// Functions/Container Statistics/F_VN_MaxElementElementwise/F_VN_MaxElementElementwise_TcVnVector2_INT

	{attribute 'TcIecLibraryType'}
	{attribute 'external_name' := 'F_VN_MaxElementElementwise_TcVnVector2_INT_GUID_51ECF3A6_4E5F_DFF9_82EE_852C7A6E0756'}
	(* Gets the element wise maximum container element. *)
	FUNCTION F_VN_MaxElementElementwise_TcVnVector2_INT : HRESULT
	VAR_INPUT
		ipContainer	:	ITcVnContainer;	(* Source container *)
	END_VAR
	VAR_IN_OUT
		aMax	:	TcVnVector2_INT;	(* Returns the requested element *)
	END_VAR
	VAR_INPUT
		hrPrev	:	HRESULT;	(* HRESULT indicating the result of previous operations (If SUCCEEDED(hrPrev) equals false, no operation is executed.) *)
	END_VAR

END_FUNCTION

// Functions/Container Statistics/F_VN_MaxElementElementwise/F_VN_MaxElementElementwise_TcVnVector2_REAL

	{attribute 'TcIecLibraryType'}
	{attribute 'external_name' := 'F_VN_MaxElementElementwise_TcVnVector2_REAL_GUID_36FF9044_FDCF_D9B2_9EF3_5D22DF14193D'}
	(* Gets the element wise maximum container element. *)
	FUNCTION F_VN_MaxElementElementwise_TcVnVector2_REAL : HRESULT
	VAR_INPUT
		ipContainer	:	ITcVnContainer;	(* Source container *)
	END_VAR
	VAR_IN_OUT
		aMax	:	TcVnVector2_REAL;	(* Returns the requested element *)
	END_VAR
	VAR_INPUT
		hrPrev	:	HRESULT;	(* HRESULT indicating the result of previous operations (If SUCCEEDED(hrPrev) equals false, no operation is executed.) *)
	END_VAR

END_FUNCTION

// Functions/Container Statistics/F_VN_MaxElementElementwise/F_VN_MaxElementElementwise_TcVnVector2_SINT

	{attribute 'TcIecLibraryType'}
	{attribute 'external_name' := 'F_VN_MaxElementElementwise_TcVnVector2_SINT_GUID_B2222E5E_8B5F_D4D8_B8B7_613F506655FE'}
	(* Gets the element wise maximum container element. *)
	FUNCTION F_VN_MaxElementElementwise_TcVnVector2_SINT : HRESULT
	VAR_INPUT
		ipContainer	:	ITcVnContainer;	(* Source container *)
	END_VAR
	VAR_IN_OUT
		aMax	:	TcVnVector2_SINT;	(* Returns the requested element *)
	END_VAR
	VAR_INPUT
		hrPrev	:	HRESULT;	(* HRESULT indicating the result of previous operations (If SUCCEEDED(hrPrev) equals false, no operation is executed.) *)
	END_VAR

END_FUNCTION

// Functions/Container Statistics/F_VN_MaxElementElementwise/F_VN_MaxElementElementwise_TcVnVector2_UINT

	{attribute 'TcIecLibraryType'}
	{attribute 'external_name' := 'F_VN_MaxElementElementwise_TcVnVector2_UINT_GUID_20FFCD90_266D_DEF6_B943_7766169A45FA'}
	(* Gets the element wise maximum container element. *)
	FUNCTION F_VN_MaxElementElementwise_TcVnVector2_UINT : HRESULT
	VAR_INPUT
		ipContainer	:	ITcVnContainer;	(* Source container *)
	END_VAR
	VAR_IN_OUT
		aMax	:	TcVnVector2_UINT;	(* Returns the requested element *)
	END_VAR
	VAR_INPUT
		hrPrev	:	HRESULT;	(* HRESULT indicating the result of previous operations (If SUCCEEDED(hrPrev) equals false, no operation is executed.) *)
	END_VAR

END_FUNCTION

// Functions/Container Statistics/F_VN_MaxElementElementwise/F_VN_MaxElementElementwise_TcVnVector2_USINT

	{attribute 'TcIecLibraryType'}
	{attribute 'external_name' := 'F_VN_MaxElementElementwise_TcVnVector2_USINT_GUID_759705D1_AC56_D8D1_B875_EB16D1D15497'}
	(* Gets the element wise maximum container element. *)
	FUNCTION F_VN_MaxElementElementwise_TcVnVector2_USINT : HRESULT
	VAR_INPUT
		ipContainer	:	ITcVnContainer;	(* Source container *)
	END_VAR
	VAR_IN_OUT
		aMax	:	TcVnVector2_USINT;	(* Returns the requested element *)
	END_VAR
	VAR_INPUT
		hrPrev	:	HRESULT;	(* HRESULT indicating the result of previous operations (If SUCCEEDED(hrPrev) equals false, no operation is executed.) *)
	END_VAR

END_FUNCTION

// Functions/Container Statistics/F_VN_MaxElementElementwise/F_VN_MaxElementElementwise_TcVnVector3_INT

	{attribute 'TcIecLibraryType'}
	{attribute 'external_name' := 'F_VN_MaxElementElementwise_TcVnVector3_INT_GUID_8201BE4F_7FA6_D4DA_A679_F7186350AEF1'}
	(* Gets the element wise maximum container element. *)
	FUNCTION F_VN_MaxElementElementwise_TcVnVector3_INT : HRESULT
	VAR_INPUT
		ipContainer	:	ITcVnContainer;	(* Source container *)
	END_VAR
	VAR_IN_OUT
		aMax	:	TcVnVector3_INT;	(* Returns the requested element *)
	END_VAR
	VAR_INPUT
		hrPrev	:	HRESULT;	(* HRESULT indicating the result of previous operations (If SUCCEEDED(hrPrev) equals false, no operation is executed.) *)
	END_VAR

END_FUNCTION

// Functions/Container Statistics/F_VN_MaxElementElementwise/F_VN_MaxElementElementwise_TcVnVector3_REAL

	{attribute 'TcIecLibraryType'}
	{attribute 'external_name' := 'F_VN_MaxElementElementwise_TcVnVector3_REAL_GUID_01B744AE_DDF1_D8D6_AD1D_2564E4DF54AD'}
	(* Gets the element wise maximum container element. *)
	FUNCTION F_VN_MaxElementElementwise_TcVnVector3_REAL : HRESULT
	VAR_INPUT
		ipContainer	:	ITcVnContainer;	(* Source container *)
	END_VAR
	VAR_IN_OUT
		aMax	:	TcVnVector3_REAL;	(* Returns the requested element *)
	END_VAR
	VAR_INPUT
		hrPrev	:	HRESULT;	(* HRESULT indicating the result of previous operations (If SUCCEEDED(hrPrev) equals false, no operation is executed.) *)
	END_VAR

END_FUNCTION

// Functions/Container Statistics/F_VN_MaxElementElementwise/F_VN_MaxElementElementwise_TcVnVector3_SINT

	{attribute 'TcIecLibraryType'}
	{attribute 'external_name' := 'F_VN_MaxElementElementwise_TcVnVector3_SINT_GUID_62FCA671_CE0E_D9DF_B91A_305D94F8EDEB'}
	(* Gets the element wise maximum container element. *)
	FUNCTION F_VN_MaxElementElementwise_TcVnVector3_SINT : HRESULT
	VAR_INPUT
		ipContainer	:	ITcVnContainer;	(* Source container *)
	END_VAR
	VAR_IN_OUT
		aMax	:	TcVnVector3_SINT;	(* Returns the requested element *)
	END_VAR
	VAR_INPUT
		hrPrev	:	HRESULT;	(* HRESULT indicating the result of previous operations (If SUCCEEDED(hrPrev) equals false, no operation is executed.) *)
	END_VAR

END_FUNCTION

// Functions/Container Statistics/F_VN_MaxElementElementwise/F_VN_MaxElementElementwise_TcVnVector3_UINT

	{attribute 'TcIecLibraryType'}
	{attribute 'external_name' := 'F_VN_MaxElementElementwise_TcVnVector3_UINT_GUID_17CA3582_D75B_D4E5_96F3_81C1A0815197'}
	(* Gets the element wise maximum container element. *)
	FUNCTION F_VN_MaxElementElementwise_TcVnVector3_UINT : HRESULT
	VAR_INPUT
		ipContainer	:	ITcVnContainer;	(* Source container *)
	END_VAR
	VAR_IN_OUT
		aMax	:	TcVnVector3_UINT;	(* Returns the requested element *)
	END_VAR
	VAR_INPUT
		hrPrev	:	HRESULT;	(* HRESULT indicating the result of previous operations (If SUCCEEDED(hrPrev) equals false, no operation is executed.) *)
	END_VAR

END_FUNCTION

// Functions/Container Statistics/F_VN_MaxElementElementwise/F_VN_MaxElementElementwise_TcVnVector3_USINT

	{attribute 'TcIecLibraryType'}
	{attribute 'external_name' := 'F_VN_MaxElementElementwise_TcVnVector3_USINT_GUID_CA4AC978_BB4E_DA6E_A59D_D0FAA5AA5CC0'}
	(* Gets the element wise maximum container element. *)
	FUNCTION F_VN_MaxElementElementwise_TcVnVector3_USINT : HRESULT
	VAR_INPUT
		ipContainer	:	ITcVnContainer;	(* Source container *)
	END_VAR
	VAR_IN_OUT
		aMax	:	TcVnVector3_USINT;	(* Returns the requested element *)
	END_VAR
	VAR_INPUT
		hrPrev	:	HRESULT;	(* HRESULT indicating the result of previous operations (If SUCCEEDED(hrPrev) equals false, no operation is executed.) *)
	END_VAR

END_FUNCTION

// Functions/Container Statistics/F_VN_MaxElementElementwise/F_VN_MaxElementElementwise_TcVnVector4_DINT

	{attribute 'TcIecLibraryType'}
	{attribute 'external_name' := 'F_VN_MaxElementElementwise_TcVnVector4_DINT_GUID_CD328B5F_53BD_D10E_830D_85DBB5B313E2'}
	(* Gets the element wise maximum container element. *)
	FUNCTION F_VN_MaxElementElementwise_TcVnVector4_DINT : HRESULT
	VAR_INPUT
		ipContainer	:	ITcVnContainer;	(* Source container *)
	END_VAR
	VAR_IN_OUT
		aMax	:	TcVnVector4_DINT;	(* Returns the requested element *)
	END_VAR
	VAR_INPUT
		hrPrev	:	HRESULT;	(* HRESULT indicating the result of previous operations (If SUCCEEDED(hrPrev) equals false, no operation is executed.) *)
	END_VAR

END_FUNCTION

// Functions/Container Statistics/F_VN_MaxElementElementwise/F_VN_MaxElementElementwise_TcVnVector4_INT

	{attribute 'TcIecLibraryType'}
	{attribute 'external_name' := 'F_VN_MaxElementElementwise_TcVnVector4_INT_GUID_1F26472A_5D0C_D30F_BDCF_211A9E9155AD'}
	(* Gets the element wise maximum container element. *)
	FUNCTION F_VN_MaxElementElementwise_TcVnVector4_INT : HRESULT
	VAR_INPUT
		ipContainer	:	ITcVnContainer;	(* Source container *)
	END_VAR
	VAR_IN_OUT
		aMax	:	TcVnVector4_INT;	(* Returns the requested element *)
	END_VAR
	VAR_INPUT
		hrPrev	:	HRESULT;	(* HRESULT indicating the result of previous operations (If SUCCEEDED(hrPrev) equals false, no operation is executed.) *)
	END_VAR

END_FUNCTION

// Functions/Container Statistics/F_VN_MaxElementElementwise/F_VN_MaxElementElementwise_TcVnVector4_LREAL

	{attribute 'TcIecLibraryType'}
	{attribute 'external_name' := 'F_VN_MaxElementElementwise_TcVnVector4_LREAL_GUID_F7067E46_8455_DE11_B5D6_36771A946BF9'}
	(* Gets the element wise maximum container element. *)
	FUNCTION F_VN_MaxElementElementwise_TcVnVector4_LREAL : HRESULT
	VAR_INPUT
		ipContainer	:	ITcVnContainer;	(* Source container *)
	END_VAR
	VAR_IN_OUT
		aMax	:	TcVnVector4_LREAL;	(* Returns the requested element *)
	END_VAR
	VAR_INPUT
		hrPrev	:	HRESULT;	(* HRESULT indicating the result of previous operations (If SUCCEEDED(hrPrev) equals false, no operation is executed.) *)
	END_VAR

END_FUNCTION

// Functions/Container Statistics/F_VN_MaxElementElementwise/F_VN_MaxElementElementwise_TcVnVector4_REAL

	{attribute 'TcIecLibraryType'}
	{attribute 'external_name' := 'F_VN_MaxElementElementwise_TcVnVector4_REAL_GUID_A7B55928_9DF9_D291_8F16_9723E5982003'}
	(* Gets the element wise maximum container element. *)
	FUNCTION F_VN_MaxElementElementwise_TcVnVector4_REAL : HRESULT
	VAR_INPUT
		ipContainer	:	ITcVnContainer;	(* Source container *)
	END_VAR
	VAR_IN_OUT
		aMax	:	TcVnVector4_REAL;	(* Returns the requested element *)
	END_VAR
	VAR_INPUT
		hrPrev	:	HRESULT;	(* HRESULT indicating the result of previous operations (If SUCCEEDED(hrPrev) equals false, no operation is executed.) *)
	END_VAR

END_FUNCTION

// Functions/Container Statistics/F_VN_MaxElementElementwise/F_VN_MaxElementElementwise_TcVnVector4_SINT

	{attribute 'TcIecLibraryType'}
	{attribute 'external_name' := 'F_VN_MaxElementElementwise_TcVnVector4_SINT_GUID_BBB783C6_087A_D40B_A284_9C1E42E427DC'}
	(* Gets the element wise maximum container element. *)
	FUNCTION F_VN_MaxElementElementwise_TcVnVector4_SINT : HRESULT
	VAR_INPUT
		ipContainer	:	ITcVnContainer;	(* Source container *)
	END_VAR
	VAR_IN_OUT
		aMax	:	TcVnVector4_SINT;	(* Returns the requested element *)
	END_VAR
	VAR_INPUT
		hrPrev	:	HRESULT;	(* HRESULT indicating the result of previous operations (If SUCCEEDED(hrPrev) equals false, no operation is executed.) *)
	END_VAR

END_FUNCTION

// Functions/Container Statistics/F_VN_MaxElementElementwise/F_VN_MaxElementElementwise_TcVnVector4_UINT

	{attribute 'TcIecLibraryType'}
	{attribute 'external_name' := 'F_VN_MaxElementElementwise_TcVnVector4_UINT_GUID_65ED7CB6_2391_D985_BD33_521B77431117'}
	(* Gets the element wise maximum container element. *)
	FUNCTION F_VN_MaxElementElementwise_TcVnVector4_UINT : HRESULT
	VAR_INPUT
		ipContainer	:	ITcVnContainer;	(* Source container *)
	END_VAR
	VAR_IN_OUT
		aMax	:	TcVnVector4_UINT;	(* Returns the requested element *)
	END_VAR
	VAR_INPUT
		hrPrev	:	HRESULT;	(* HRESULT indicating the result of previous operations (If SUCCEEDED(hrPrev) equals false, no operation is executed.) *)
	END_VAR

END_FUNCTION

// Functions/Container Statistics/F_VN_MaxElementElementwise/F_VN_MaxElementElementwise_TcVnVector4_USINT

	{attribute 'TcIecLibraryType'}
	{attribute 'external_name' := 'F_VN_MaxElementElementwise_TcVnVector4_USINT_GUID_9C34A78C_F853_D377_9C12_528CEB462408'}
	(* Gets the element wise maximum container element. *)
	FUNCTION F_VN_MaxElementElementwise_TcVnVector4_USINT : HRESULT
	VAR_INPUT
		ipContainer	:	ITcVnContainer;	(* Source container *)
	END_VAR
	VAR_IN_OUT
		aMax	:	TcVnVector4_USINT;	(* Returns the requested element *)
	END_VAR
	VAR_INPUT
		hrPrev	:	HRESULT;	(* HRESULT indicating the result of previous operations (If SUCCEEDED(hrPrev) equals false, no operation is executed.) *)
	END_VAR

END_FUNCTION

// Functions/Container Statistics/F_VN_MaxElementElementwise/F_VN_MaxElementElementwise_UDINT

	{attribute 'TcIecLibraryType'}
	{attribute 'external_name' := 'F_VN_MaxElementElementwise_UDINT_GUID_2F4B8B8C_C3F6_DAC4_AE5F_3F8AE16BC0CF'}
	(* Gets the element wise maximum container element. *)
	FUNCTION F_VN_MaxElementElementwise_UDINT : HRESULT
	VAR_INPUT
		ipContainer	:	ITcVnContainer;	(* Source container *)
	END_VAR
	VAR_IN_OUT
		nMax	:	UDINT;	(* Returns the requested element *)
	END_VAR
	VAR_INPUT
		hrPrev	:	HRESULT;	(* HRESULT indicating the result of previous operations (If SUCCEEDED(hrPrev) equals false, no operation is executed.) *)
	END_VAR

END_FUNCTION

// Functions/Container Statistics/F_VN_MaxElementElementwise/F_VN_MaxElementElementwise_UINT

	{attribute 'TcIecLibraryType'}
	{attribute 'external_name' := 'F_VN_MaxElementElementwise_UINT_GUID_2C850313_EE79_D952_8816_C7A292497C14'}
	(* Gets the element wise maximum container element. *)
	FUNCTION F_VN_MaxElementElementwise_UINT : HRESULT
	VAR_INPUT
		ipContainer	:	ITcVnContainer;	(* Source container *)
	END_VAR
	VAR_IN_OUT
		nMax	:	UINT;	(* Returns the requested element *)
	END_VAR
	VAR_INPUT
		hrPrev	:	HRESULT;	(* HRESULT indicating the result of previous operations (If SUCCEEDED(hrPrev) equals false, no operation is executed.) *)
	END_VAR

END_FUNCTION

// Functions/Container Statistics/F_VN_MaxElementElementwise/F_VN_MaxElementElementwise_ULINT

	{attribute 'TcIecLibraryType'}
	{attribute 'external_name' := 'F_VN_MaxElementElementwise_ULINT_GUID_79575080_6C4D_DE0A_A408_669186C9D1B9'}
	(* Gets the element wise maximum container element. *)
	FUNCTION F_VN_MaxElementElementwise_ULINT : HRESULT
	VAR_INPUT
		ipContainer	:	ITcVnContainer;	(* Source container *)
	END_VAR
	VAR_IN_OUT
		nMax	:	ULINT;	(* Returns the requested element *)
	END_VAR
	VAR_INPUT
		hrPrev	:	HRESULT;	(* HRESULT indicating the result of previous operations (If SUCCEEDED(hrPrev) equals false, no operation is executed.) *)
	END_VAR

END_FUNCTION

// Functions/Container Statistics/F_VN_MaxElementElementwise/F_VN_MaxElementElementwise_USINT

	{attribute 'TcIecLibraryType'}
	{attribute 'external_name' := 'F_VN_MaxElementElementwise_USINT_GUID_65E5FDF1_4B0E_DAE8_B45E_43E6CAE87A8D'}
	(* Gets the element wise maximum container element. *)
	FUNCTION F_VN_MaxElementElementwise_USINT : HRESULT
	VAR_INPUT
		ipContainer	:	ITcVnContainer;	(* Source container *)
	END_VAR
	VAR_IN_OUT
		nMax	:	USINT;	(* Returns the requested element *)
	END_VAR
	VAR_INPUT
		hrPrev	:	HRESULT;	(* HRESULT indicating the result of previous operations (If SUCCEEDED(hrPrev) equals false, no operation is executed.) *)
	END_VAR

END_FUNCTION

// Functions/Container Statistics/F_VN_MedianElementElementwise/F_VN_MedianElementElementwise_DINT

	{attribute 'TcIecLibraryType'}
	{attribute 'external_name' := 'F_VN_MedianElementElementwise_DINT_GUID_29AA868C_E552_D86B_BF6B_18030732A5CC'}
	(* Gets the element wise median container element. *)
	FUNCTION F_VN_MedianElementElementwise_DINT : HRESULT
	VAR_INPUT
		ipContainer	:	ITcVnContainer;	(* Source container *)
	END_VAR
	VAR_IN_OUT
		nMedian	:	DINT;	(* Returns the requested element *)
	END_VAR
	VAR_INPUT
		hrPrev	:	HRESULT;	(* HRESULT indicating the result of previous operations (If SUCCEEDED(hrPrev) equals false, no operation is executed.) *)
	END_VAR

END_FUNCTION

// Functions/Container Statistics/F_VN_MedianElementElementwise/F_VN_MedianElementElementwise_INT

	{attribute 'TcIecLibraryType'}
	{attribute 'external_name' := 'F_VN_MedianElementElementwise_INT_GUID_CB0AC784_E2F3_DD60_B341_B4C0DD83E5BD'}
	(* Gets the element wise median container element. *)
	FUNCTION F_VN_MedianElementElementwise_INT : HRESULT
	VAR_INPUT
		ipContainer	:	ITcVnContainer;	(* Source container *)
	END_VAR
	VAR_IN_OUT
		nMedian	:	INT;	(* Returns the requested element *)
	END_VAR
	VAR_INPUT
		hrPrev	:	HRESULT;	(* HRESULT indicating the result of previous operations (If SUCCEEDED(hrPrev) equals false, no operation is executed.) *)
	END_VAR

END_FUNCTION

// Functions/Container Statistics/F_VN_MedianElementElementwise/F_VN_MedianElementElementwise_LREAL

	{attribute 'TcIecLibraryType'}
	{attribute 'external_name' := 'F_VN_MedianElementElementwise_LREAL_GUID_B5611EAF_9AFA_D3DE_9C03_D3DC20ACA830'}
	(* Gets the element wise median container element. *)
	FUNCTION F_VN_MedianElementElementwise_LREAL : HRESULT
	VAR_INPUT
		ipContainer	:	ITcVnContainer;	(* Source container *)
	END_VAR
	VAR_IN_OUT
		fMedian	:	LREAL;	(* Returns the requested element *)
	END_VAR
	VAR_INPUT
		hrPrev	:	HRESULT;	(* HRESULT indicating the result of previous operations (If SUCCEEDED(hrPrev) equals false, no operation is executed.) *)
	END_VAR

END_FUNCTION

// Functions/Container Statistics/F_VN_MedianElementElementwise/F_VN_MedianElementElementwise_REAL

	{attribute 'TcIecLibraryType'}
	{attribute 'external_name' := 'F_VN_MedianElementElementwise_REAL_GUID_21DEF917_9EFB_D3A8_BB2F_45041A3E4378'}
	(* Gets the element wise median container element. *)
	FUNCTION F_VN_MedianElementElementwise_REAL : HRESULT
	VAR_INPUT
		ipContainer	:	ITcVnContainer;	(* Source container *)
	END_VAR
	VAR_IN_OUT
		fMedian	:	REAL;	(* Returns the requested element *)
	END_VAR
	VAR_INPUT
		hrPrev	:	HRESULT;	(* HRESULT indicating the result of previous operations (If SUCCEEDED(hrPrev) equals false, no operation is executed.) *)
	END_VAR

END_FUNCTION

// Functions/Container Statistics/F_VN_MedianElementElementwise/F_VN_MedianElementElementwise_SINT

	{attribute 'TcIecLibraryType'}
	{attribute 'external_name' := 'F_VN_MedianElementElementwise_SINT_GUID_A76B5E76_04B8_D72A_96E3_B134E306B796'}
	(* Gets the element wise median container element. *)
	FUNCTION F_VN_MedianElementElementwise_SINT : HRESULT
	VAR_INPUT
		ipContainer	:	ITcVnContainer;	(* Source container *)
	END_VAR
	VAR_IN_OUT
		nMedian	:	SINT;	(* Returns the requested element *)
	END_VAR
	VAR_INPUT
		hrPrev	:	HRESULT;	(* HRESULT indicating the result of previous operations (If SUCCEEDED(hrPrev) equals false, no operation is executed.) *)
	END_VAR

END_FUNCTION

// Functions/Container Statistics/F_VN_MedianElementElementwise/F_VN_MedianElementElementwise_TcVnPoint2_DINT

	{attribute 'TcIecLibraryType'}
	{attribute 'external_name' := 'F_VN_MedianElementElementwise_TcVnPoint2_DINT_GUID_A3592C7D_4475_D8E1_B303_A13CD5FC38FB'}
	(* Gets the element wise median container element. *)
	FUNCTION F_VN_MedianElementElementwise_TcVnPoint2_DINT : HRESULT
	VAR_INPUT
		ipContainer	:	ITcVnContainer;	(* Source container *)
	END_VAR
	VAR_IN_OUT
		aMedian	:	TcVnPoint2_DINT;	(* Returns the requested element *)
	END_VAR
	VAR_INPUT
		hrPrev	:	HRESULT;	(* HRESULT indicating the result of previous operations (If SUCCEEDED(hrPrev) equals false, no operation is executed.) *)
	END_VAR

END_FUNCTION

// Functions/Container Statistics/F_VN_MedianElementElementwise/F_VN_MedianElementElementwise_TcVnPoint2_LREAL

	{attribute 'TcIecLibraryType'}
	{attribute 'external_name' := 'F_VN_MedianElementElementwise_TcVnPoint2_LREAL_GUID_58AAC7EB_5ADE_DF64_AAA7_24D37077B229'}
	(* Gets the element wise median container element. *)
	FUNCTION F_VN_MedianElementElementwise_TcVnPoint2_LREAL : HRESULT
	VAR_INPUT
		ipContainer	:	ITcVnContainer;	(* Source container *)
	END_VAR
	VAR_IN_OUT
		aMedian	:	TcVnPoint2_LREAL;	(* Returns the requested element *)
	END_VAR
	VAR_INPUT
		hrPrev	:	HRESULT;	(* HRESULT indicating the result of previous operations (If SUCCEEDED(hrPrev) equals false, no operation is executed.) *)
	END_VAR

END_FUNCTION

// Functions/Container Statistics/F_VN_MedianElementElementwise/F_VN_MedianElementElementwise_TcVnPoint2_REAL

	{attribute 'TcIecLibraryType'}
	{attribute 'external_name' := 'F_VN_MedianElementElementwise_TcVnPoint2_REAL_GUID_F85373B6_2943_D6B1_9993_6D4DB4D57329'}
	(* Gets the element wise median container element. *)
	FUNCTION F_VN_MedianElementElementwise_TcVnPoint2_REAL : HRESULT
	VAR_INPUT
		ipContainer	:	ITcVnContainer;	(* Source container *)
	END_VAR
	VAR_IN_OUT
		aMedian	:	TcVnPoint2_REAL;	(* Returns the requested element *)
	END_VAR
	VAR_INPUT
		hrPrev	:	HRESULT;	(* HRESULT indicating the result of previous operations (If SUCCEEDED(hrPrev) equals false, no operation is executed.) *)
	END_VAR

END_FUNCTION

// Functions/Container Statistics/F_VN_MedianElementElementwise/F_VN_MedianElementElementwise_TcVnPoint3_LREAL

	{attribute 'TcIecLibraryType'}
	{attribute 'external_name' := 'F_VN_MedianElementElementwise_TcVnPoint3_LREAL_GUID_F14A33BF_2275_D80A_AC45_515904B471A2'}
	(* Gets the element wise median container element. *)
	FUNCTION F_VN_MedianElementElementwise_TcVnPoint3_LREAL : HRESULT
	VAR_INPUT
		ipContainer	:	ITcVnContainer;	(* Source container *)
	END_VAR
	VAR_IN_OUT
		aMedian	:	TcVnPoint3_LREAL;	(* Returns the requested element *)
	END_VAR
	VAR_INPUT
		hrPrev	:	HRESULT;	(* HRESULT indicating the result of previous operations (If SUCCEEDED(hrPrev) equals false, no operation is executed.) *)
	END_VAR

END_FUNCTION

// Functions/Container Statistics/F_VN_MedianElementElementwise/F_VN_MedianElementElementwise_TcVnPoint3_REAL

	{attribute 'TcIecLibraryType'}
	{attribute 'external_name' := 'F_VN_MedianElementElementwise_TcVnPoint3_REAL_GUID_756F28F9_77FF_DB99_A3DB_C5C4C4331351'}
	(* Gets the element wise median container element. *)
	FUNCTION F_VN_MedianElementElementwise_TcVnPoint3_REAL : HRESULT
	VAR_INPUT
		ipContainer	:	ITcVnContainer;	(* Source container *)
	END_VAR
	VAR_IN_OUT
		aMedian	:	TcVnPoint3_REAL;	(* Returns the requested element *)
	END_VAR
	VAR_INPUT
		hrPrev	:	HRESULT;	(* HRESULT indicating the result of previous operations (If SUCCEEDED(hrPrev) equals false, no operation is executed.) *)
	END_VAR

END_FUNCTION

// Functions/Container Statistics/F_VN_MedianElementElementwise/F_VN_MedianElementElementwise_TcVnVector2_DINT

	{attribute 'TcIecLibraryType'}
	{attribute 'external_name' := 'F_VN_MedianElementElementwise_TcVnVector2_DINT_GUID_8E473526_A7CC_DFC3_9E5F_288766125041'}
	(* Gets the element wise median container element. *)
	FUNCTION F_VN_MedianElementElementwise_TcVnVector2_DINT : HRESULT
	VAR_INPUT
		ipContainer	:	ITcVnContainer;	(* Source container *)
	END_VAR
	VAR_IN_OUT
		aMedian	:	TcVnVector2_DINT;	(* Returns the requested element *)
	END_VAR
	VAR_INPUT
		hrPrev	:	HRESULT;	(* HRESULT indicating the result of previous operations (If SUCCEEDED(hrPrev) equals false, no operation is executed.) *)
	END_VAR

END_FUNCTION

// Functions/Container Statistics/F_VN_MedianElementElementwise/F_VN_MedianElementElementwise_TcVnVector2_INT

	{attribute 'TcIecLibraryType'}
	{attribute 'external_name' := 'F_VN_MedianElementElementwise_TcVnVector2_INT_GUID_5BDD346F_B29E_DEEB_A174_03D5BCDD966C'}
	(* Gets the element wise median container element. *)
	FUNCTION F_VN_MedianElementElementwise_TcVnVector2_INT : HRESULT
	VAR_INPUT
		ipContainer	:	ITcVnContainer;	(* Source container *)
	END_VAR
	VAR_IN_OUT
		aMedian	:	TcVnVector2_INT;	(* Returns the requested element *)
	END_VAR
	VAR_INPUT
		hrPrev	:	HRESULT;	(* HRESULT indicating the result of previous operations (If SUCCEEDED(hrPrev) equals false, no operation is executed.) *)
	END_VAR

END_FUNCTION

// Functions/Container Statistics/F_VN_MedianElementElementwise/F_VN_MedianElementElementwise_TcVnVector2_REAL

	{attribute 'TcIecLibraryType'}
	{attribute 'external_name' := 'F_VN_MedianElementElementwise_TcVnVector2_REAL_GUID_86E9BF9E_E3F9_D74F_9617_EB2C03F6B6E3'}
	(* Gets the element wise median container element. *)
	FUNCTION F_VN_MedianElementElementwise_TcVnVector2_REAL : HRESULT
	VAR_INPUT
		ipContainer	:	ITcVnContainer;	(* Source container *)
	END_VAR
	VAR_IN_OUT
		aMedian	:	TcVnVector2_REAL;	(* Returns the requested element *)
	END_VAR
	VAR_INPUT
		hrPrev	:	HRESULT;	(* HRESULT indicating the result of previous operations (If SUCCEEDED(hrPrev) equals false, no operation is executed.) *)
	END_VAR

END_FUNCTION

// Functions/Container Statistics/F_VN_MedianElementElementwise/F_VN_MedianElementElementwise_TcVnVector2_SINT

	{attribute 'TcIecLibraryType'}
	{attribute 'external_name' := 'F_VN_MedianElementElementwise_TcVnVector2_SINT_GUID_FF27191B_A2BB_DF95_854B_1FD1821A0F7E'}
	(* Gets the element wise median container element. *)
	FUNCTION F_VN_MedianElementElementwise_TcVnVector2_SINT : HRESULT
	VAR_INPUT
		ipContainer	:	ITcVnContainer;	(* Source container *)
	END_VAR
	VAR_IN_OUT
		aMedian	:	TcVnVector2_SINT;	(* Returns the requested element *)
	END_VAR
	VAR_INPUT
		hrPrev	:	HRESULT;	(* HRESULT indicating the result of previous operations (If SUCCEEDED(hrPrev) equals false, no operation is executed.) *)
	END_VAR

END_FUNCTION

// Functions/Container Statistics/F_VN_MedianElementElementwise/F_VN_MedianElementElementwise_TcVnVector2_UINT

	{attribute 'TcIecLibraryType'}
	{attribute 'external_name' := 'F_VN_MedianElementElementwise_TcVnVector2_UINT_GUID_705877EF_7F8F_DC5B_A99E_E66FED4F7A28'}
	(* Gets the element wise median container element. *)
	FUNCTION F_VN_MedianElementElementwise_TcVnVector2_UINT : HRESULT
	VAR_INPUT
		ipContainer	:	ITcVnContainer;	(* Source container *)
	END_VAR
	VAR_IN_OUT
		aMedian	:	TcVnVector2_UINT;	(* Returns the requested element *)
	END_VAR
	VAR_INPUT
		hrPrev	:	HRESULT;	(* HRESULT indicating the result of previous operations (If SUCCEEDED(hrPrev) equals false, no operation is executed.) *)
	END_VAR

END_FUNCTION

// Functions/Container Statistics/F_VN_MedianElementElementwise/F_VN_MedianElementElementwise_TcVnVector2_USINT

	{attribute 'TcIecLibraryType'}
	{attribute 'external_name' := 'F_VN_MedianElementElementwise_TcVnVector2_USINT_GUID_25701AD9_252E_DC2D_9926_E17D1B44381C'}
	(* Gets the element wise median container element. *)
	FUNCTION F_VN_MedianElementElementwise_TcVnVector2_USINT : HRESULT
	VAR_INPUT
		ipContainer	:	ITcVnContainer;	(* Source container *)
	END_VAR
	VAR_IN_OUT
		aMedian	:	TcVnVector2_USINT;	(* Returns the requested element *)
	END_VAR
	VAR_INPUT
		hrPrev	:	HRESULT;	(* HRESULT indicating the result of previous operations (If SUCCEEDED(hrPrev) equals false, no operation is executed.) *)
	END_VAR

END_FUNCTION

// Functions/Container Statistics/F_VN_MedianElementElementwise/F_VN_MedianElementElementwise_TcVnVector3_INT

	{attribute 'TcIecLibraryType'}
	{attribute 'external_name' := 'F_VN_MedianElementElementwise_TcVnVector3_INT_GUID_4CD6D63F_F997_D2F3_AB3B_4A33E5647F84'}
	(* Gets the element wise median container element. *)
	FUNCTION F_VN_MedianElementElementwise_TcVnVector3_INT : HRESULT
	VAR_INPUT
		ipContainer	:	ITcVnContainer;	(* Source container *)
	END_VAR
	VAR_IN_OUT
		aMedian	:	TcVnVector3_INT;	(* Returns the requested element *)
	END_VAR
	VAR_INPUT
		hrPrev	:	HRESULT;	(* HRESULT indicating the result of previous operations (If SUCCEEDED(hrPrev) equals false, no operation is executed.) *)
	END_VAR

END_FUNCTION

// Functions/Container Statistics/F_VN_MedianElementElementwise/F_VN_MedianElementElementwise_TcVnVector3_REAL

	{attribute 'TcIecLibraryType'}
	{attribute 'external_name' := 'F_VN_MedianElementElementwise_TcVnVector3_REAL_GUID_4E994DD7_D9B7_DE3E_932B_AC8B406F870C'}
	(* Gets the element wise median container element. *)
	FUNCTION F_VN_MedianElementElementwise_TcVnVector3_REAL : HRESULT
	VAR_INPUT
		ipContainer	:	ITcVnContainer;	(* Source container *)
	END_VAR
	VAR_IN_OUT
		aMedian	:	TcVnVector3_REAL;	(* Returns the requested element *)
	END_VAR
	VAR_INPUT
		hrPrev	:	HRESULT;	(* HRESULT indicating the result of previous operations (If SUCCEEDED(hrPrev) equals false, no operation is executed.) *)
	END_VAR

END_FUNCTION

// Functions/Container Statistics/F_VN_MedianElementElementwise/F_VN_MedianElementElementwise_TcVnVector3_SINT

	{attribute 'TcIecLibraryType'}
	{attribute 'external_name' := 'F_VN_MedianElementElementwise_TcVnVector3_SINT_GUID_9137D501_0F28_D22B_853D_E2549CAB39F0'}
	(* Gets the element wise median container element. *)
	FUNCTION F_VN_MedianElementElementwise_TcVnVector3_SINT : HRESULT
	VAR_INPUT
		ipContainer	:	ITcVnContainer;	(* Source container *)
	END_VAR
	VAR_IN_OUT
		aMedian	:	TcVnVector3_SINT;	(* Returns the requested element *)
	END_VAR
	VAR_INPUT
		hrPrev	:	HRESULT;	(* HRESULT indicating the result of previous operations (If SUCCEEDED(hrPrev) equals false, no operation is executed.) *)
	END_VAR

END_FUNCTION

// Functions/Container Statistics/F_VN_MedianElementElementwise/F_VN_MedianElementElementwise_TcVnVector3_UINT

	{attribute 'TcIecLibraryType'}
	{attribute 'external_name' := 'F_VN_MedianElementElementwise_TcVnVector3_UINT_GUID_A8DF8F4C_462A_D898_950A_55B3BB3E2024'}
	(* Gets the element wise median container element. *)
	FUNCTION F_VN_MedianElementElementwise_TcVnVector3_UINT : HRESULT
	VAR_INPUT
		ipContainer	:	ITcVnContainer;	(* Source container *)
	END_VAR
	VAR_IN_OUT
		aMedian	:	TcVnVector3_UINT;	(* Returns the requested element *)
	END_VAR
	VAR_INPUT
		hrPrev	:	HRESULT;	(* HRESULT indicating the result of previous operations (If SUCCEEDED(hrPrev) equals false, no operation is executed.) *)
	END_VAR

END_FUNCTION

// Functions/Container Statistics/F_VN_MedianElementElementwise/F_VN_MedianElementElementwise_TcVnVector3_USINT

	{attribute 'TcIecLibraryType'}
	{attribute 'external_name' := 'F_VN_MedianElementElementwise_TcVnVector3_USINT_GUID_0C8F98E8_0B46_D076_9A4C_AEBC34133C5E'}
	(* Gets the element wise median container element. *)
	FUNCTION F_VN_MedianElementElementwise_TcVnVector3_USINT : HRESULT
	VAR_INPUT
		ipContainer	:	ITcVnContainer;	(* Source container *)
	END_VAR
	VAR_IN_OUT
		aMedian	:	TcVnVector3_USINT;	(* Returns the requested element *)
	END_VAR
	VAR_INPUT
		hrPrev	:	HRESULT;	(* HRESULT indicating the result of previous operations (If SUCCEEDED(hrPrev) equals false, no operation is executed.) *)
	END_VAR

END_FUNCTION

// Functions/Container Statistics/F_VN_MedianElementElementwise/F_VN_MedianElementElementwise_TcVnVector4_DINT

	{attribute 'TcIecLibraryType'}
	{attribute 'external_name' := 'F_VN_MedianElementElementwise_TcVnVector4_DINT_GUID_6FADAB1A_0169_D530_9009_CC67F58ABF30'}
	(* Gets the element wise median container element. *)
	FUNCTION F_VN_MedianElementElementwise_TcVnVector4_DINT : HRESULT
	VAR_INPUT
		ipContainer	:	ITcVnContainer;	(* Source container *)
	END_VAR
	VAR_IN_OUT
		aMedian	:	TcVnVector4_DINT;	(* Returns the requested element *)
	END_VAR
	VAR_INPUT
		hrPrev	:	HRESULT;	(* HRESULT indicating the result of previous operations (If SUCCEEDED(hrPrev) equals false, no operation is executed.) *)
	END_VAR

END_FUNCTION

// Functions/Container Statistics/F_VN_MedianElementElementwise/F_VN_MedianElementElementwise_TcVnVector4_INT

	{attribute 'TcIecLibraryType'}
	{attribute 'external_name' := 'F_VN_MedianElementElementwise_TcVnVector4_INT_GUID_547BAD9B_6F7A_DD0B_8790_02EDB713B258'}
	(* Gets the element wise median container element. *)
	FUNCTION F_VN_MedianElementElementwise_TcVnVector4_INT : HRESULT
	VAR_INPUT
		ipContainer	:	ITcVnContainer;	(* Source container *)
	END_VAR
	VAR_IN_OUT
		aMedian	:	TcVnVector4_INT;	(* Returns the requested element *)
	END_VAR
	VAR_INPUT
		hrPrev	:	HRESULT;	(* HRESULT indicating the result of previous operations (If SUCCEEDED(hrPrev) equals false, no operation is executed.) *)
	END_VAR

END_FUNCTION

// Functions/Container Statistics/F_VN_MedianElementElementwise/F_VN_MedianElementElementwise_TcVnVector4_LREAL

	{attribute 'TcIecLibraryType'}
	{attribute 'external_name' := 'F_VN_MedianElementElementwise_TcVnVector4_LREAL_GUID_626602F4_5A0A_DEBF_AF13_43F5508850CD'}
	(* Gets the element wise median container element. *)
	FUNCTION F_VN_MedianElementElementwise_TcVnVector4_LREAL : HRESULT
	VAR_INPUT
		ipContainer	:	ITcVnContainer;	(* Source container *)
	END_VAR
	VAR_IN_OUT
		aMedian	:	TcVnVector4_LREAL;	(* Returns the requested element *)
	END_VAR
	VAR_INPUT
		hrPrev	:	HRESULT;	(* HRESULT indicating the result of previous operations (If SUCCEEDED(hrPrev) equals false, no operation is executed.) *)
	END_VAR

END_FUNCTION

// Functions/Container Statistics/F_VN_MedianElementElementwise/F_VN_MedianElementElementwise_TcVnVector4_REAL

	{attribute 'TcIecLibraryType'}
	{attribute 'external_name' := 'F_VN_MedianElementElementwise_TcVnVector4_REAL_GUID_49F75D51_3181_DA08_9B3B_68B99A9DF7AE'}
	(* Gets the element wise median container element. *)
	FUNCTION F_VN_MedianElementElementwise_TcVnVector4_REAL : HRESULT
	VAR_INPUT
		ipContainer	:	ITcVnContainer;	(* Source container *)
	END_VAR
	VAR_IN_OUT
		aMedian	:	TcVnVector4_REAL;	(* Returns the requested element *)
	END_VAR
	VAR_INPUT
		hrPrev	:	HRESULT;	(* HRESULT indicating the result of previous operations (If SUCCEEDED(hrPrev) equals false, no operation is executed.) *)
	END_VAR

END_FUNCTION

// Functions/Container Statistics/F_VN_MedianElementElementwise/F_VN_MedianElementElementwise_TcVnVector4_SINT

	{attribute 'TcIecLibraryType'}
	{attribute 'external_name' := 'F_VN_MedianElementElementwise_TcVnVector4_SINT_GUID_61695308_1194_D30C_87B3_CD47BB5B616F'}
	(* Gets the element wise median container element. *)
	FUNCTION F_VN_MedianElementElementwise_TcVnVector4_SINT : HRESULT
	VAR_INPUT
		ipContainer	:	ITcVnContainer;	(* Source container *)
	END_VAR
	VAR_IN_OUT
		aMedian	:	TcVnVector4_SINT;	(* Returns the requested element *)
	END_VAR
	VAR_INPUT
		hrPrev	:	HRESULT;	(* HRESULT indicating the result of previous operations (If SUCCEEDED(hrPrev) equals false, no operation is executed.) *)
	END_VAR

END_FUNCTION

// Functions/Container Statistics/F_VN_MedianElementElementwise/F_VN_MedianElementElementwise_TcVnVector4_UINT

	{attribute 'TcIecLibraryType'}
	{attribute 'external_name' := 'F_VN_MedianElementElementwise_TcVnVector4_UINT_GUID_04BDB311_7306_D375_920D_775A084C28E2'}
	(* Gets the element wise median container element. *)
	FUNCTION F_VN_MedianElementElementwise_TcVnVector4_UINT : HRESULT
	VAR_INPUT
		ipContainer	:	ITcVnContainer;	(* Source container *)
	END_VAR
	VAR_IN_OUT
		aMedian	:	TcVnVector4_UINT;	(* Returns the requested element *)
	END_VAR
	VAR_INPUT
		hrPrev	:	HRESULT;	(* HRESULT indicating the result of previous operations (If SUCCEEDED(hrPrev) equals false, no operation is executed.) *)
	END_VAR

END_FUNCTION

// Functions/Container Statistics/F_VN_MedianElementElementwise/F_VN_MedianElementElementwise_TcVnVector4_USINT

	{attribute 'TcIecLibraryType'}
	{attribute 'external_name' := 'F_VN_MedianElementElementwise_TcVnVector4_USINT_GUID_C6120573_4FCC_DD80_AD43_4ABD35A8D98B'}
	(* Gets the element wise median container element. *)
	FUNCTION F_VN_MedianElementElementwise_TcVnVector4_USINT : HRESULT
	VAR_INPUT
		ipContainer	:	ITcVnContainer;	(* Source container *)
	END_VAR
	VAR_IN_OUT
		aMedian	:	TcVnVector4_USINT;	(* Returns the requested element *)
	END_VAR
	VAR_INPUT
		hrPrev	:	HRESULT;	(* HRESULT indicating the result of previous operations (If SUCCEEDED(hrPrev) equals false, no operation is executed.) *)
	END_VAR

END_FUNCTION

// Functions/Container Statistics/F_VN_MedianElementElementwise/F_VN_MedianElementElementwise_UDINT

	{attribute 'TcIecLibraryType'}
	{attribute 'external_name' := 'F_VN_MedianElementElementwise_UDINT_GUID_9BC7BF91_3125_D729_9768_84FE886C888D'}
	(* Gets the element wise median container element. *)
	FUNCTION F_VN_MedianElementElementwise_UDINT : HRESULT
	VAR_INPUT
		ipContainer	:	ITcVnContainer;	(* Source container *)
	END_VAR
	VAR_IN_OUT
		nMedian	:	UDINT;	(* Returns the requested element *)
	END_VAR
	VAR_INPUT
		hrPrev	:	HRESULT;	(* HRESULT indicating the result of previous operations (If SUCCEEDED(hrPrev) equals false, no operation is executed.) *)
	END_VAR

END_FUNCTION

// Functions/Container Statistics/F_VN_MedianElementElementwise/F_VN_MedianElementElementwise_UINT

	{attribute 'TcIecLibraryType'}
	{attribute 'external_name' := 'F_VN_MedianElementElementwise_UINT_GUID_AA7E04F5_27DD_D1E9_89BB_71FE2A03EF73'}
	(* Gets the element wise median container element. *)
	FUNCTION F_VN_MedianElementElementwise_UINT : HRESULT
	VAR_INPUT
		ipContainer	:	ITcVnContainer;	(* Source container *)
	END_VAR
	VAR_IN_OUT
		nMedian	:	UINT;	(* Returns the requested element *)
	END_VAR
	VAR_INPUT
		hrPrev	:	HRESULT;	(* HRESULT indicating the result of previous operations (If SUCCEEDED(hrPrev) equals false, no operation is executed.) *)
	END_VAR

END_FUNCTION

// Functions/Container Statistics/F_VN_MedianElementElementwise/F_VN_MedianElementElementwise_ULINT

	{attribute 'TcIecLibraryType'}
	{attribute 'external_name' := 'F_VN_MedianElementElementwise_ULINT_GUID_8ECFBFA6_0E43_DAD1_AF9F_464DAE11C1ED'}
	(* Gets the element wise median container element. *)
	FUNCTION F_VN_MedianElementElementwise_ULINT : HRESULT
	VAR_INPUT
		ipContainer	:	ITcVnContainer;	(* Source container *)
	END_VAR
	VAR_IN_OUT
		nMedian	:	ULINT;	(* Returns the requested element *)
	END_VAR
	VAR_INPUT
		hrPrev	:	HRESULT;	(* HRESULT indicating the result of previous operations (If SUCCEEDED(hrPrev) equals false, no operation is executed.) *)
	END_VAR

END_FUNCTION

// Functions/Container Statistics/F_VN_MedianElementElementwise/F_VN_MedianElementElementwise_USINT

	{attribute 'TcIecLibraryType'}
	{attribute 'external_name' := 'F_VN_MedianElementElementwise_USINT_GUID_2994888C_8833_D8FA_BA03_E55B76F2506A'}
	(* Gets the element wise median container element. *)
	FUNCTION F_VN_MedianElementElementwise_USINT : HRESULT
	VAR_INPUT
		ipContainer	:	ITcVnContainer;	(* Source container *)
	END_VAR
	VAR_IN_OUT
		nMedian	:	USINT;	(* Returns the requested element *)
	END_VAR
	VAR_INPUT
		hrPrev	:	HRESULT;	(* HRESULT indicating the result of previous operations (If SUCCEEDED(hrPrev) equals false, no operation is executed.) *)
	END_VAR

END_FUNCTION

// Functions/Container Statistics/F_VN_MinElementElementwise/F_VN_MinElementElementwise_DINT

	{attribute 'TcIecLibraryType'}
	{attribute 'external_name' := 'F_VN_MinElementElementwise_DINT_GUID_7E567114_9BD1_D305_87D1_88AF602BEA2D'}
	(* Gets the element wise minimum container element. *)
	FUNCTION F_VN_MinElementElementwise_DINT : HRESULT
	VAR_INPUT
		ipContainer	:	ITcVnContainer;	(* Source container *)
	END_VAR
	VAR_IN_OUT
		nMin	:	DINT;	(* Returns the requested element *)
	END_VAR
	VAR_INPUT
		hrPrev	:	HRESULT;	(* HRESULT indicating the result of previous operations (If SUCCEEDED(hrPrev) equals false, no operation is executed.) *)
	END_VAR

END_FUNCTION

// Functions/Container Statistics/F_VN_MinElementElementwise/F_VN_MinElementElementwise_INT

	{attribute 'TcIecLibraryType'}
	{attribute 'external_name' := 'F_VN_MinElementElementwise_INT_GUID_0BB9518D_66CC_D115_B745_E5695DFD31B0'}
	(* Gets the element wise minimum container element. *)
	FUNCTION F_VN_MinElementElementwise_INT : HRESULT
	VAR_INPUT
		ipContainer	:	ITcVnContainer;	(* Source container *)
	END_VAR
	VAR_IN_OUT
		nMin	:	INT;	(* Returns the requested element *)
	END_VAR
	VAR_INPUT
		hrPrev	:	HRESULT;	(* HRESULT indicating the result of previous operations (If SUCCEEDED(hrPrev) equals false, no operation is executed.) *)
	END_VAR

END_FUNCTION

// Functions/Container Statistics/F_VN_MinElementElementwise/F_VN_MinElementElementwise_LREAL

	{attribute 'TcIecLibraryType'}
	{attribute 'external_name' := 'F_VN_MinElementElementwise_LREAL_GUID_C1D5880C_C085_D406_8F8C_640347E2EC83'}
	(* Gets the element wise minimum container element. *)
	FUNCTION F_VN_MinElementElementwise_LREAL : HRESULT
	VAR_INPUT
		ipContainer	:	ITcVnContainer;	(* Source container *)
	END_VAR
	VAR_IN_OUT
		fMin	:	LREAL;	(* Returns the requested element *)
	END_VAR
	VAR_INPUT
		hrPrev	:	HRESULT;	(* HRESULT indicating the result of previous operations (If SUCCEEDED(hrPrev) equals false, no operation is executed.) *)
	END_VAR

END_FUNCTION

// Functions/Container Statistics/F_VN_MinElementElementwise/F_VN_MinElementElementwise_REAL

	{attribute 'TcIecLibraryType'}
	{attribute 'external_name' := 'F_VN_MinElementElementwise_REAL_GUID_450605AD_BDF8_DB97_BA29_50E9A007428F'}
	(* Gets the element wise minimum container element. *)
	FUNCTION F_VN_MinElementElementwise_REAL : HRESULT
	VAR_INPUT
		ipContainer	:	ITcVnContainer;	(* Source container *)
	END_VAR
	VAR_IN_OUT
		fMin	:	REAL;	(* Returns the requested element *)
	END_VAR
	VAR_INPUT
		hrPrev	:	HRESULT;	(* HRESULT indicating the result of previous operations (If SUCCEEDED(hrPrev) equals false, no operation is executed.) *)
	END_VAR

END_FUNCTION

// Functions/Container Statistics/F_VN_MinElementElementwise/F_VN_MinElementElementwise_SINT

	{attribute 'TcIecLibraryType'}
	{attribute 'external_name' := 'F_VN_MinElementElementwise_SINT_GUID_2E0DA260_F5E9_DFCE_81FD_D87F2E028328'}
	(* Gets the element wise minimum container element. *)
	FUNCTION F_VN_MinElementElementwise_SINT : HRESULT
	VAR_INPUT
		ipContainer	:	ITcVnContainer;	(* Source container *)
	END_VAR
	VAR_IN_OUT
		nMin	:	SINT;	(* Returns the requested element *)
	END_VAR
	VAR_INPUT
		hrPrev	:	HRESULT;	(* HRESULT indicating the result of previous operations (If SUCCEEDED(hrPrev) equals false, no operation is executed.) *)
	END_VAR

END_FUNCTION

// Functions/Container Statistics/F_VN_MinElementElementwise/F_VN_MinElementElementwise_TcVnPoint2_DINT

	{attribute 'TcIecLibraryType'}
	{attribute 'external_name' := 'F_VN_MinElementElementwise_TcVnPoint2_DINT_GUID_0EC94E3E_0D59_DE54_86BC_2993576C6132'}
	(* Gets the element wise minimum container element. *)
	FUNCTION F_VN_MinElementElementwise_TcVnPoint2_DINT : HRESULT
	VAR_INPUT
		ipContainer	:	ITcVnContainer;	(* Source container *)
	END_VAR
	VAR_IN_OUT
		aMin	:	TcVnPoint2_DINT;	(* Returns the requested element *)
	END_VAR
	VAR_INPUT
		hrPrev	:	HRESULT;	(* HRESULT indicating the result of previous operations (If SUCCEEDED(hrPrev) equals false, no operation is executed.) *)
	END_VAR

END_FUNCTION

// Functions/Container Statistics/F_VN_MinElementElementwise/F_VN_MinElementElementwise_TcVnPoint2_LREAL

	{attribute 'TcIecLibraryType'}
	{attribute 'external_name' := 'F_VN_MinElementElementwise_TcVnPoint2_LREAL_GUID_9AFC6C99_4848_D8F3_B855_368B34F740F2'}
	(* Gets the element wise minimum container element. *)
	FUNCTION F_VN_MinElementElementwise_TcVnPoint2_LREAL : HRESULT
	VAR_INPUT
		ipContainer	:	ITcVnContainer;	(* Source container *)
	END_VAR
	VAR_IN_OUT
		aMin	:	TcVnPoint2_LREAL;	(* Returns the requested element *)
	END_VAR
	VAR_INPUT
		hrPrev	:	HRESULT;	(* HRESULT indicating the result of previous operations (If SUCCEEDED(hrPrev) equals false, no operation is executed.) *)
	END_VAR

END_FUNCTION

// Functions/Container Statistics/F_VN_MinElementElementwise/F_VN_MinElementElementwise_TcVnPoint2_REAL

	{attribute 'TcIecLibraryType'}
	{attribute 'external_name' := 'F_VN_MinElementElementwise_TcVnPoint2_REAL_GUID_7AC6B98C_169A_DF8C_964B_4FAA29A72F57'}
	(* Gets the element wise minimum container element. *)
	FUNCTION F_VN_MinElementElementwise_TcVnPoint2_REAL : HRESULT
	VAR_INPUT
		ipContainer	:	ITcVnContainer;	(* Source container *)
	END_VAR
	VAR_IN_OUT
		aMin	:	TcVnPoint2_REAL;	(* Returns the requested element *)
	END_VAR
	VAR_INPUT
		hrPrev	:	HRESULT;	(* HRESULT indicating the result of previous operations (If SUCCEEDED(hrPrev) equals false, no operation is executed.) *)
	END_VAR

END_FUNCTION

// Functions/Container Statistics/F_VN_MinElementElementwise/F_VN_MinElementElementwise_TcVnPoint3_LREAL

	{attribute 'TcIecLibraryType'}
	{attribute 'external_name' := 'F_VN_MinElementElementwise_TcVnPoint3_LREAL_GUID_B02BC3B2_A0BF_D7E4_8FF2_614514F5F69D'}
	(* Gets the element wise minimum container element. *)
	FUNCTION F_VN_MinElementElementwise_TcVnPoint3_LREAL : HRESULT
	VAR_INPUT
		ipContainer	:	ITcVnContainer;	(* Source container *)
	END_VAR
	VAR_IN_OUT
		aMin	:	TcVnPoint3_LREAL;	(* Returns the requested element *)
	END_VAR
	VAR_INPUT
		hrPrev	:	HRESULT;	(* HRESULT indicating the result of previous operations (If SUCCEEDED(hrPrev) equals false, no operation is executed.) *)
	END_VAR

END_FUNCTION

// Functions/Container Statistics/F_VN_MinElementElementwise/F_VN_MinElementElementwise_TcVnPoint3_REAL

	{attribute 'TcIecLibraryType'}
	{attribute 'external_name' := 'F_VN_MinElementElementwise_TcVnPoint3_REAL_GUID_166E82CB_FBD6_D924_BFB7_F50CA7DCAC72'}
	(* Gets the element wise minimum container element. *)
	FUNCTION F_VN_MinElementElementwise_TcVnPoint3_REAL : HRESULT
	VAR_INPUT
		ipContainer	:	ITcVnContainer;	(* Source container *)
	END_VAR
	VAR_IN_OUT
		aMin	:	TcVnPoint3_REAL;	(* Returns the requested element *)
	END_VAR
	VAR_INPUT
		hrPrev	:	HRESULT;	(* HRESULT indicating the result of previous operations (If SUCCEEDED(hrPrev) equals false, no operation is executed.) *)
	END_VAR

END_FUNCTION

// Functions/Container Statistics/F_VN_MinElementElementwise/F_VN_MinElementElementwise_TcVnVector2_DINT

	{attribute 'TcIecLibraryType'}
	{attribute 'external_name' := 'F_VN_MinElementElementwise_TcVnVector2_DINT_GUID_4AF02B0D_6242_D42D_9C65_E65E956B738B'}
	(* Gets the element wise minimum container element. *)
	FUNCTION F_VN_MinElementElementwise_TcVnVector2_DINT : HRESULT
	VAR_INPUT
		ipContainer	:	ITcVnContainer;	(* Source container *)
	END_VAR
	VAR_IN_OUT
		aMin	:	TcVnVector2_DINT;	(* Returns the requested element *)
	END_VAR
	VAR_INPUT
		hrPrev	:	HRESULT;	(* HRESULT indicating the result of previous operations (If SUCCEEDED(hrPrev) equals false, no operation is executed.) *)
	END_VAR

END_FUNCTION

// Functions/Container Statistics/F_VN_MinElementElementwise/F_VN_MinElementElementwise_TcVnVector2_INT

	{attribute 'TcIecLibraryType'}
	{attribute 'external_name' := 'F_VN_MinElementElementwise_TcVnVector2_INT_GUID_519E35CF_AFCF_D40A_9DCC_7890A636C2FC'}
	(* Gets the element wise minimum container element. *)
	FUNCTION F_VN_MinElementElementwise_TcVnVector2_INT : HRESULT
	VAR_INPUT
		ipContainer	:	ITcVnContainer;	(* Source container *)
	END_VAR
	VAR_IN_OUT
		aMin	:	TcVnVector2_INT;	(* Returns the requested element *)
	END_VAR
	VAR_INPUT
		hrPrev	:	HRESULT;	(* HRESULT indicating the result of previous operations (If SUCCEEDED(hrPrev) equals false, no operation is executed.) *)
	END_VAR

END_FUNCTION

// Functions/Container Statistics/F_VN_MinElementElementwise/F_VN_MinElementElementwise_TcVnVector2_REAL

	{attribute 'TcIecLibraryType'}
	{attribute 'external_name' := 'F_VN_MinElementElementwise_TcVnVector2_REAL_GUID_852C686C_8B53_DEB2_85E9_0E846F82CC51'}
	(* Gets the element wise minimum container element. *)
	FUNCTION F_VN_MinElementElementwise_TcVnVector2_REAL : HRESULT
	VAR_INPUT
		ipContainer	:	ITcVnContainer;	(* Source container *)
	END_VAR
	VAR_IN_OUT
		aMin	:	TcVnVector2_REAL;	(* Returns the requested element *)
	END_VAR
	VAR_INPUT
		hrPrev	:	HRESULT;	(* HRESULT indicating the result of previous operations (If SUCCEEDED(hrPrev) equals false, no operation is executed.) *)
	END_VAR

END_FUNCTION

// Functions/Container Statistics/F_VN_MinElementElementwise/F_VN_MinElementElementwise_TcVnVector2_SINT

	{attribute 'TcIecLibraryType'}
	{attribute 'external_name' := 'F_VN_MinElementElementwise_TcVnVector2_SINT_GUID_45CD3985_C6EF_DBC6_B7FF_EA5FD0C160D8'}
	(* Gets the element wise minimum container element. *)
	FUNCTION F_VN_MinElementElementwise_TcVnVector2_SINT : HRESULT
	VAR_INPUT
		ipContainer	:	ITcVnContainer;	(* Source container *)
	END_VAR
	VAR_IN_OUT
		aMin	:	TcVnVector2_SINT;	(* Returns the requested element *)
	END_VAR
	VAR_INPUT
		hrPrev	:	HRESULT;	(* HRESULT indicating the result of previous operations (If SUCCEEDED(hrPrev) equals false, no operation is executed.) *)
	END_VAR

END_FUNCTION

// Functions/Container Statistics/F_VN_MinElementElementwise/F_VN_MinElementElementwise_TcVnVector2_UINT

	{attribute 'TcIecLibraryType'}
	{attribute 'external_name' := 'F_VN_MinElementElementwise_TcVnVector2_UINT_GUID_82DD13C1_BC80_DB01_A28F_B92C7A2F1C96'}
	(* Gets the element wise minimum container element. *)
	FUNCTION F_VN_MinElementElementwise_TcVnVector2_UINT : HRESULT
	VAR_INPUT
		ipContainer	:	ITcVnContainer;	(* Source container *)
	END_VAR
	VAR_IN_OUT
		aMin	:	TcVnVector2_UINT;	(* Returns the requested element *)
	END_VAR
	VAR_INPUT
		hrPrev	:	HRESULT;	(* HRESULT indicating the result of previous operations (If SUCCEEDED(hrPrev) equals false, no operation is executed.) *)
	END_VAR

END_FUNCTION

// Functions/Container Statistics/F_VN_MinElementElementwise/F_VN_MinElementElementwise_TcVnVector2_USINT

	{attribute 'TcIecLibraryType'}
	{attribute 'external_name' := 'F_VN_MinElementElementwise_TcVnVector2_USINT_GUID_D4C45077_8215_D85D_AC8B_F8E314D4D048'}
	(* Gets the element wise minimum container element. *)
	FUNCTION F_VN_MinElementElementwise_TcVnVector2_USINT : HRESULT
	VAR_INPUT
		ipContainer	:	ITcVnContainer;	(* Source container *)
	END_VAR
	VAR_IN_OUT
		aMin	:	TcVnVector2_USINT;	(* Returns the requested element *)
	END_VAR
	VAR_INPUT
		hrPrev	:	HRESULT;	(* HRESULT indicating the result of previous operations (If SUCCEEDED(hrPrev) equals false, no operation is executed.) *)
	END_VAR

END_FUNCTION

// Functions/Container Statistics/F_VN_MinElementElementwise/F_VN_MinElementElementwise_TcVnVector3_INT

	{attribute 'TcIecLibraryType'}
	{attribute 'external_name' := 'F_VN_MinElementElementwise_TcVnVector3_INT_GUID_003F395B_72A0_D2D0_BC5C_704EE36651C3'}
	(* Gets the element wise minimum container element. *)
	FUNCTION F_VN_MinElementElementwise_TcVnVector3_INT : HRESULT
	VAR_INPUT
		ipContainer	:	ITcVnContainer;	(* Source container *)
	END_VAR
	VAR_IN_OUT
		aMin	:	TcVnVector3_INT;	(* Returns the requested element *)
	END_VAR
	VAR_INPUT
		hrPrev	:	HRESULT;	(* HRESULT indicating the result of previous operations (If SUCCEEDED(hrPrev) equals false, no operation is executed.) *)
	END_VAR

END_FUNCTION

// Functions/Container Statistics/F_VN_MinElementElementwise/F_VN_MinElementElementwise_TcVnVector3_REAL

	{attribute 'TcIecLibraryType'}
	{attribute 'external_name' := 'F_VN_MinElementElementwise_TcVnVector3_REAL_GUID_CCFCB828_1C38_DAF0_9900_DD6020B17524'}
	(* Gets the element wise minimum container element. *)
	FUNCTION F_VN_MinElementElementwise_TcVnVector3_REAL : HRESULT
	VAR_INPUT
		ipContainer	:	ITcVnContainer;	(* Source container *)
	END_VAR
	VAR_IN_OUT
		aMin	:	TcVnVector3_REAL;	(* Returns the requested element *)
	END_VAR
	VAR_INPUT
		hrPrev	:	HRESULT;	(* HRESULT indicating the result of previous operations (If SUCCEEDED(hrPrev) equals false, no operation is executed.) *)
	END_VAR

END_FUNCTION

// Functions/Container Statistics/F_VN_MinElementElementwise/F_VN_MinElementElementwise_TcVnVector3_SINT

	{attribute 'TcIecLibraryType'}
	{attribute 'external_name' := 'F_VN_MinElementElementwise_TcVnVector3_SINT_GUID_60BB9A8F_4E3E_D660_A368_6B00FE16B99F'}
	(* Gets the element wise minimum container element. *)
	FUNCTION F_VN_MinElementElementwise_TcVnVector3_SINT : HRESULT
	VAR_INPUT
		ipContainer	:	ITcVnContainer;	(* Source container *)
	END_VAR
	VAR_IN_OUT
		aMin	:	TcVnVector3_SINT;	(* Returns the requested element *)
	END_VAR
	VAR_INPUT
		hrPrev	:	HRESULT;	(* HRESULT indicating the result of previous operations (If SUCCEEDED(hrPrev) equals false, no operation is executed.) *)
	END_VAR

END_FUNCTION

// Functions/Container Statistics/F_VN_MinElementElementwise/F_VN_MinElementElementwise_TcVnVector3_UINT

	{attribute 'TcIecLibraryType'}
	{attribute 'external_name' := 'F_VN_MinElementElementwise_TcVnVector3_UINT_GUID_32AB90CF_8AF3_DC7D_BB5D_2E61BC6B1430'}
	(* Gets the element wise minimum container element. *)
	FUNCTION F_VN_MinElementElementwise_TcVnVector3_UINT : HRESULT
	VAR_INPUT
		ipContainer	:	ITcVnContainer;	(* Source container *)
	END_VAR
	VAR_IN_OUT
		aMin	:	TcVnVector3_UINT;	(* Returns the requested element *)
	END_VAR
	VAR_INPUT
		hrPrev	:	HRESULT;	(* HRESULT indicating the result of previous operations (If SUCCEEDED(hrPrev) equals false, no operation is executed.) *)
	END_VAR

END_FUNCTION

// Functions/Container Statistics/F_VN_MinElementElementwise/F_VN_MinElementElementwise_TcVnVector3_USINT

	{attribute 'TcIecLibraryType'}
	{attribute 'external_name' := 'F_VN_MinElementElementwise_TcVnVector3_USINT_GUID_6CE7D88D_9B81_D1BC_B929_63928ECEF2A3'}
	(* Gets the element wise minimum container element. *)
	FUNCTION F_VN_MinElementElementwise_TcVnVector3_USINT : HRESULT
	VAR_INPUT
		ipContainer	:	ITcVnContainer;	(* Source container *)
	END_VAR
	VAR_IN_OUT
		aMin	:	TcVnVector3_USINT;	(* Returns the requested element *)
	END_VAR
	VAR_INPUT
		hrPrev	:	HRESULT;	(* HRESULT indicating the result of previous operations (If SUCCEEDED(hrPrev) equals false, no operation is executed.) *)
	END_VAR

END_FUNCTION

// Functions/Container Statistics/F_VN_MinElementElementwise/F_VN_MinElementElementwise_TcVnVector4_DINT

	{attribute 'TcIecLibraryType'}
	{attribute 'external_name' := 'F_VN_MinElementElementwise_TcVnVector4_DINT_GUID_4A4F38C3_6AA6_DCD9_9449_56537B19CC16'}
	(* Gets the element wise minimum container element. *)
	FUNCTION F_VN_MinElementElementwise_TcVnVector4_DINT : HRESULT
	VAR_INPUT
		ipContainer	:	ITcVnContainer;	(* Source container *)
	END_VAR
	VAR_IN_OUT
		aMin	:	TcVnVector4_DINT;	(* Returns the requested element *)
	END_VAR
	VAR_INPUT
		hrPrev	:	HRESULT;	(* HRESULT indicating the result of previous operations (If SUCCEEDED(hrPrev) equals false, no operation is executed.) *)
	END_VAR

END_FUNCTION

// Functions/Container Statistics/F_VN_MinElementElementwise/F_VN_MinElementElementwise_TcVnVector4_INT

	{attribute 'TcIecLibraryType'}
	{attribute 'external_name' := 'F_VN_MinElementElementwise_TcVnVector4_INT_GUID_F46A250E_E6A1_DC56_9D11_B98E3F59D525'}
	(* Gets the element wise minimum container element. *)
	FUNCTION F_VN_MinElementElementwise_TcVnVector4_INT : HRESULT
	VAR_INPUT
		ipContainer	:	ITcVnContainer;	(* Source container *)
	END_VAR
	VAR_IN_OUT
		aMin	:	TcVnVector4_INT;	(* Returns the requested element *)
	END_VAR
	VAR_INPUT
		hrPrev	:	HRESULT;	(* HRESULT indicating the result of previous operations (If SUCCEEDED(hrPrev) equals false, no operation is executed.) *)
	END_VAR

END_FUNCTION

// Functions/Container Statistics/F_VN_MinElementElementwise/F_VN_MinElementElementwise_TcVnVector4_LREAL

	{attribute 'TcIecLibraryType'}
	{attribute 'external_name' := 'F_VN_MinElementElementwise_TcVnVector4_LREAL_GUID_CC843590_6FD0_DB17_BFBC_2283C26E6041'}
	(* Gets the element wise minimum container element. *)
	FUNCTION F_VN_MinElementElementwise_TcVnVector4_LREAL : HRESULT
	VAR_INPUT
		ipContainer	:	ITcVnContainer;	(* Source container *)
	END_VAR
	VAR_IN_OUT
		aMin	:	TcVnVector4_LREAL;	(* Returns the requested element *)
	END_VAR
	VAR_INPUT
		hrPrev	:	HRESULT;	(* HRESULT indicating the result of previous operations (If SUCCEEDED(hrPrev) equals false, no operation is executed.) *)
	END_VAR

END_FUNCTION

// Functions/Container Statistics/F_VN_MinElementElementwise/F_VN_MinElementElementwise_TcVnVector4_REAL

	{attribute 'TcIecLibraryType'}
	{attribute 'external_name' := 'F_VN_MinElementElementwise_TcVnVector4_REAL_GUID_0B3FFE65_262F_D136_9ACC_7C737C28E6C7'}
	(* Gets the element wise minimum container element. *)
	FUNCTION F_VN_MinElementElementwise_TcVnVector4_REAL : HRESULT
	VAR_INPUT
		ipContainer	:	ITcVnContainer;	(* Source container *)
	END_VAR
	VAR_IN_OUT
		aMin	:	TcVnVector4_REAL;	(* Returns the requested element *)
	END_VAR
	VAR_INPUT
		hrPrev	:	HRESULT;	(* HRESULT indicating the result of previous operations (If SUCCEEDED(hrPrev) equals false, no operation is executed.) *)
	END_VAR

END_FUNCTION

// Functions/Container Statistics/F_VN_MinElementElementwise/F_VN_MinElementElementwise_TcVnVector4_SINT

	{attribute 'TcIecLibraryType'}
	{attribute 'external_name' := 'F_VN_MinElementElementwise_TcVnVector4_SINT_GUID_131F6433_3F24_D7B7_9C79_869216C8F48D'}
	(* Gets the element wise minimum container element. *)
	FUNCTION F_VN_MinElementElementwise_TcVnVector4_SINT : HRESULT
	VAR_INPUT
		ipContainer	:	ITcVnContainer;	(* Source container *)
	END_VAR
	VAR_IN_OUT
		aMin	:	TcVnVector4_SINT;	(* Returns the requested element *)
	END_VAR
	VAR_INPUT
		hrPrev	:	HRESULT;	(* HRESULT indicating the result of previous operations (If SUCCEEDED(hrPrev) equals false, no operation is executed.) *)
	END_VAR

END_FUNCTION

// Functions/Container Statistics/F_VN_MinElementElementwise/F_VN_MinElementElementwise_TcVnVector4_UINT

	{attribute 'TcIecLibraryType'}
	{attribute 'external_name' := 'F_VN_MinElementElementwise_TcVnVector4_UINT_GUID_DCC4190A_0954_D4FA_A1F1_9A79B4CCEE16'}
	(* Gets the element wise minimum container element. *)
	FUNCTION F_VN_MinElementElementwise_TcVnVector4_UINT : HRESULT
	VAR_INPUT
		ipContainer	:	ITcVnContainer;	(* Source container *)
	END_VAR
	VAR_IN_OUT
		aMin	:	TcVnVector4_UINT;	(* Returns the requested element *)
	END_VAR
	VAR_INPUT
		hrPrev	:	HRESULT;	(* HRESULT indicating the result of previous operations (If SUCCEEDED(hrPrev) equals false, no operation is executed.) *)
	END_VAR

END_FUNCTION

// Functions/Container Statistics/F_VN_MinElementElementwise/F_VN_MinElementElementwise_TcVnVector4_USINT

	{attribute 'TcIecLibraryType'}
	{attribute 'external_name' := 'F_VN_MinElementElementwise_TcVnVector4_USINT_GUID_7BDE3AC2_7BE7_DCE9_8DCC_9DB720D63FC3'}
	(* Gets the element wise minimum container element. *)
	FUNCTION F_VN_MinElementElementwise_TcVnVector4_USINT : HRESULT
	VAR_INPUT
		ipContainer	:	ITcVnContainer;	(* Source container *)
	END_VAR
	VAR_IN_OUT
		aMin	:	TcVnVector4_USINT;	(* Returns the requested element *)
	END_VAR
	VAR_INPUT
		hrPrev	:	HRESULT;	(* HRESULT indicating the result of previous operations (If SUCCEEDED(hrPrev) equals false, no operation is executed.) *)
	END_VAR

END_FUNCTION

// Functions/Container Statistics/F_VN_MinElementElementwise/F_VN_MinElementElementwise_UDINT

	{attribute 'TcIecLibraryType'}
	{attribute 'external_name' := 'F_VN_MinElementElementwise_UDINT_GUID_70D63C8E_595B_DBA6_BC42_A2C00435489D'}
	(* Gets the element wise minimum container element. *)
	FUNCTION F_VN_MinElementElementwise_UDINT : HRESULT
	VAR_INPUT
		ipContainer	:	ITcVnContainer;	(* Source container *)
	END_VAR
	VAR_IN_OUT
		nMin	:	UDINT;	(* Returns the requested element *)
	END_VAR
	VAR_INPUT
		hrPrev	:	HRESULT;	(* HRESULT indicating the result of previous operations (If SUCCEEDED(hrPrev) equals false, no operation is executed.) *)
	END_VAR

END_FUNCTION

// Functions/Container Statistics/F_VN_MinElementElementwise/F_VN_MinElementElementwise_UINT

	{attribute 'TcIecLibraryType'}
	{attribute 'external_name' := 'F_VN_MinElementElementwise_UINT_GUID_71116108_5AC8_D1E9_8B5F_49056B04AF8D'}
	(* Gets the element wise minimum container element. *)
	FUNCTION F_VN_MinElementElementwise_UINT : HRESULT
	VAR_INPUT
		ipContainer	:	ITcVnContainer;	(* Source container *)
	END_VAR
	VAR_IN_OUT
		nMin	:	UINT;	(* Returns the requested element *)
	END_VAR
	VAR_INPUT
		hrPrev	:	HRESULT;	(* HRESULT indicating the result of previous operations (If SUCCEEDED(hrPrev) equals false, no operation is executed.) *)
	END_VAR

END_FUNCTION

// Functions/Container Statistics/F_VN_MinElementElementwise/F_VN_MinElementElementwise_ULINT

	{attribute 'TcIecLibraryType'}
	{attribute 'external_name' := 'F_VN_MinElementElementwise_ULINT_GUID_E03F40D3_6F1A_D514_B486_5AB15DF41ECC'}
	(* Gets the element wise minimum container element. *)
	FUNCTION F_VN_MinElementElementwise_ULINT : HRESULT
	VAR_INPUT
		ipContainer	:	ITcVnContainer;	(* Source container *)
	END_VAR
	VAR_IN_OUT
		nMin	:	ULINT;	(* Returns the requested element *)
	END_VAR
	VAR_INPUT
		hrPrev	:	HRESULT;	(* HRESULT indicating the result of previous operations (If SUCCEEDED(hrPrev) equals false, no operation is executed.) *)
	END_VAR

END_FUNCTION

// Functions/Container Statistics/F_VN_MinElementElementwise/F_VN_MinElementElementwise_USINT

	{attribute 'TcIecLibraryType'}
	{attribute 'external_name' := 'F_VN_MinElementElementwise_USINT_GUID_3031C9D5_DB9A_D95A_8A10_64F60244185A'}
	(* Gets the element wise minimum container element. *)
	FUNCTION F_VN_MinElementElementwise_USINT : HRESULT
	VAR_INPUT
		ipContainer	:	ITcVnContainer;	(* Source container *)
	END_VAR
	VAR_IN_OUT
		nMin	:	USINT;	(* Returns the requested element *)
	END_VAR
	VAR_INPUT
		hrPrev	:	HRESULT;	(* HRESULT indicating the result of previous operations (If SUCCEEDED(hrPrev) equals false, no operation is executed.) *)
	END_VAR

END_FUNCTION
